(* IEC 61131-3 sources: AXOpen/src/components.ur.robotics/app/src, 2 files *)

(* ---- configuration.st ---- *)
USING AXOpen.Components.Ur.Robotics;

CONFIGURATION MyConfiguration
    TASK Main(Interval := T#10ms, Priority := 1);
    PROGRAM P1 WITH Main: MyProgram;

    VAR_GLOBAL
        {S7.extern=ReadWrite}
        sandbox : SandboxContext;
        {S7.extern=ReadWrite}
        documentation : DocumentationContext;
        {S7.extern=ReadWrite}
        _rtc : AXOpen.S71500.Rtc;
    END_VAR

END_CONFIGURATION

(* ---- program.st ---- *)
USING AXOpen.Components.Ur.Robotics;

PROGRAM MyProgram
    VAR_EXTERNAL
        sandbox : SandboxContext;
        documentation : DocumentationContext;
        _rtc : AXOpen.S71500.Rtc;
    END_VAR

    sandbox.Run();
    sandbox.InjectRtc(_rtc);

    documentation.Run();
    documentation.InjectRtc(_rtc);
END_PROGRAM
